# B&R Automation Studio project Kontrol (part 3)

#### Cyclic.st
```iecst
PROGRAM _CYCLIC

    IF NOT PgsTagValid(TagManager.ident) THEN
        RETURN;
    END_IF

	cm0985Meter();

    phaseFault(
        Enable  := TRUE,
        Ph1     := cm0985Meter.Ug1,
        Ph2     := cm0985Meter.Ug2,
        Ph3     := cm0985Meter.Ug3
    );

(*******************************************************
****************** Circuit Breaker  ********************
*******************************************************)
    avr.DigInputs.Online := CB52.st.closed;
    gov.DigInputs.Online := CB52.st.closed;

(******************************************************)
    //Reset
    IF A65.di.reset THEN
        //A65.di.reset        := FALSE;
        avr.DigInputs.Reset := TRUE;
		gov.DigInputs.Reset := TRUE;
		//Reset to Auto Mode
		//gov.DigInputs.Auto  := TRUE;
		//avr.DigInputs.Auto  := TRUE;
    END_IF;

    IF NOT A65.di.remote THEN
        //GOV
        gov.DigInputs.Start     := A65.di.gov_enable;
        gov.DigInputs.Stop      := NOT A65.di.gov_enable;
        gov.DigInputs.Unload    := A65.di.gov_unload;
		gov.DigInputs.RefUp		:= A65.di.gov_up;
		gov.DigInputs.RefDown	:= A65.di.gov_down;
        IF A65.di.gov_ctrl_pwr_enable THEN
            gov.CtrlOnline  := PGS_GOV_CA_PWR;
        ELSE
            gov.CtrlOnline  := PGS_GOV_CA_HZ_1;
        END_IF;

        //AVR
		A65.di.avr_unload		:= A65.di.gov_unload;
        avr.DigInputs.Start     := A65.di.avr_enable;
        avr.DigInputs.Stop      := NOT A65.di.avr_enable;
        avr.DigInputs.Unload    := A65.di.avr_unload;
		avr.DigInputs.RefUp		:= A65.di.avr_ref_up;
		avr.DigInputs.RefDown	:= A65.di.avr_ref_down;

        IF A65.di.avr_ctrl_qm_enable    THEN
            avr.CtrlOnline  := PGS_AVR_CA_QM;
        ELSIF  A65.di.avr_ctrl_pf_enable THEN
            avr.CtrlOnline  := PGS_AVR_CA_PF;
        ELSE
            avr.CtrlOnline  := PGS_AVR_CA_UM_1;
        END_IF;

    END_IF;

    (******************************************************)

	//TRIP
	IF A65.di.avr_trip THEN
        avr.DigInputs.Stop := TRUE;
    END_IF;
    IF A65.di.gov_trip THEN
        gov.DigInputs.Stop := TRUE;
    END_IF;

	//Meters

    //Icc ==> fix 4-20mA
    scale_if.x1 := 4.0;
    scale_if.x2 := 20.0;
    if_input	:= IfAvg * 16.0 / 32767.0 + 4.0;

    scale_if(
        x   := if_input,
        y1  := SysPar.Gen.IfMin,
        y2  := SysPar.Gen.IfMax
    );
	meter.In.If := scale_if.y;

	//Vcc ==> fix 4-20mA
    scale_uf.x1 := 4.0;
    scale_uf.x2 := 20.0;
	uf_input	:= UfAvg * 16.0 / 32767.0 + 4.0;
    scale_uf(
        x   := uf_input,
        y1  := SysPar.Gen.UfMin,
        y2  := SysPar.Gen.UfMax
    );
	meter.In.Uf := scale_uf.y;

	filter_uf( x := meter.In.Uf );
    //Ub
    IF cm0985Main.Enable3phase THEN
        meter.In.Ub := (cm0985Meter.Un12 + cm0985Meter.Un23 + cm0985Meter.Un31) / 3;
    ELSE
        meter.In.Ub := cm0985Meter.Un12;
    END_IF;
	//Um
	IF NOT phaseFault.Fault1 AND NOT phaseFault.Fault2 AND NOT phaseFault.Fault3 THEN
        meter.In.Um 	:=  cm0985Meter.Ug;
    ELSIF phaseFault.Fault1 AND NOT phaseFault.Fault2 AND NOT phaseFault.Fault3 THEN
        meter.In.Um 	:=  cm0985Meter.Ug23;
    ELSIF NOT phaseFault.Fault1 AND phaseFault.Fault2 AND NOT phaseFault.Fault3 THEN
        meter.In.Um 	:=  cm0985Meter.Ug31;
    ELSIF NOT phaseFault.Fault1 AND NOT phaseFault.Fault2 AND phaseFault.Fault3 THEN
        meter.In.Um 	:=  cm0985Meter.Ug12;
    ELSE
        meter.In.Um     :=  phaseFault.Phm * SQRT(3);
    END_IF

	meter.In.Im		:= cm0985Meter.Ig;
	IF meter.In.Um < 5 THEN
		meter.In.Fm		:= 0.0;
		meter.In.PF		:= 1.0;
	ELSE
		meter.In.Fm		:= cm0985Meter.Fg;
		meter.In.PF		:= cm0985Meter.PFg;
	END_IF;
	meter.In.Pm		:= cm0985Meter.Pg;
	meter.In.Qm		:= cm0985Meter.Qg;
	meter.In.Sm		:= cm0985Meter.Sg;

    rpm1(ppr := REAL_TO_INT(SysPar.Gen.PPR1));
    filter_rpm1.IN := rpm1.Output;
	filter_rpm1();

    rpm2(ppr := REAL_TO_INT(SysPar.Gen.PPR2));
    IF SysPar.Gen.PPR2 <> 0 THEN
		filter_rpm2.IN := rpm2.Output;
	ELSE
		filter_rpm2.IN := 0.0;
	END_IF;
    filter_rpm2();

	IF filter_rpm1.OUT > filter_rpm2.OUT THEN
	    meter.In.Rot := filter_rpm1.OUT;
    ELSE
	    meter.In.Rot := filter_rpm2.OUT;
    END_IF;

	IF SysPar.Gen.PPR2 <> 0 THEN
		A65.do.rpm_fault := ( ABS(filter_rpm1.OUT - filter_rpm2.OUT) / meter.Base.Rot ) > 0.05;
	ELSE
		A65.do.rpm_fault := FALSE;
	END_IF;
	meter       ();

	//Position
    //pos1 - ==> fix 4-20mA
	pos1_input	    := INT_TO_REAL(A65.ai.pos1) * 16.0 / 32767.0 + 4.0;
	filter_pos1(IN:=pos1_input);
    scale_pos1(
        x   := filter_pos1.OUT,
		x1  := SysPar.Gen.Pos1_0p,
        x2  := SysPar.Gen.Pos1_100p
    );
	pos1.PosIn	:= scale_pos1.y;

    pos2_input	    := INT_TO_REAL(A65.ai.pos2) * 16.0 / 32767.0 + 4.0;
    scale_pos2(
        x   := pos2_input,
		x1  := SysPar.Gen.Pos2_0p,
		x2  := SysPar.Gen.Pos2_100p
	);
	pos2.PosIn	:= scale_pos2.y;

    pos3_input	    := INT_TO_REAL(A65.ai.pos3) * 16.0 / 32767.0 + 4.0;
    scale_pos3(
        x   := pos3_input,
		x1  := SysPar.Gen.Pos3_0p,
		x2  := SysPar.Gen.Pos3_100p
	);
    pos3.PosIn := scale_pos3.y;

	//Syncronizer
    IF A65.di.remote THEN
        cm0985IO.do.SyncSlip    := SysUpdate.EnableSync;
        cm0985IO.do.SyncDeadBus := SysUpdate.EnableDeadBus AND NOT SysUpdate.EnableSync;
    ELSE
        cm0985IO.do.SyncSlip    := A65.di.sync_enable AND NOT CB52.st.closed;
        cm0985IO.do.SyncDeadBus := A65.di.dead_bus_enable AND NOT CB52.st.closed AND NOT A65.di.sync_enable;
    END_IF;
	A65.do.sync_enabled     := cm0985IO.do.SyncSlip OR cm0985IO.do.SyncDeadBus;
    IF cm0985IO.do.SyncSlip THEN
		IF cm0985Meter.dAngle > 15 AND cm0985Meter.dAngle < 345 THEN
			gov.SetPoints.fastSetHz := (cm0985Meter.Fs1 / meter.Base.Fm) * 1.001;
		ELSE
			gov.SetPoints.fastSetHz := cm0985Meter.Fs1 / meter.Base.Fm;
		END_IF;
		avr.SetPoints.fastSetUm := meter.Out.Ub;
	END_IF;

//=======================================================================
//=====	Para maior estabilidade do controle de potência	=================
//=======================================================================
	// Filtro da leitura da potência para estabilizar o sinal
	IF meter.Out.Pm <> 0 THEN
		filter_pwr(IN:=meter.Out.Pm);
	ELSE
		filter_pwr(IN:=0.0001);
	END_IF;
	// Verifica se a diferença em módulo da potência é menor que 1.5%
	IF  ABS(filter_pwr.OUT - gov.SetPoints.fastSetPwr) < gov.Parameter.CtrlAuto.CaPwr.Kdp
		// Verifica se a diferença em módulo do controle é menor que 2%
	AND ABS(1 - gov.SetPoints.fastSetHz) < 0.02	THEN
		// Se a deadband do PID for diferente, aplica deadband
		IF gov.Parameter.CtrlAuto.CaPwr.PID.db <> gov.Parameter.CtrlAuto.CaPwr.Kdp THEN
			gov.Parameter.CtrlAuto.CaPwr.PID.Update		:= TRUE;
			gov.Parameter.CtrlAuto.CaPwr.PIDHz.Update	:= TRUE;
		END_IF;
		gov.Parameter.CtrlAuto.CaPwr.PID.db		:= gov.Parameter.CtrlAuto.CaPwr.Kdp;
		gov.Parameter.CtrlAuto.CaPwr.PIDHz.db	:= gov.Parameter.CtrlAuto.CaPwr.Kdp;
	ELSE
		// Se a deadband do PID for diferente, desaplica deadband
		IF gov.Parameter.CtrlAuto.CaPwr.PID.db <> 0.00 THEN
			gov.Parameter.CtrlAuto.CaPwr.PID.Update	:= TRUE;
			gov.Parameter.CtrlAuto.CaPwr.PIDHz.Update	:= TRUE;
		END_IF;
		gov.Parameter.CtrlAuto.CaPwr.PID.db		:= 0.00;
		gov.Parameter.CtrlAuto.CaPwr.PIDHz.db	:= 0.00;
	END_IF;

	pwr_tp(IN:= CB52.st.closed, PT:=T#2s);
	IF pwr_tp.Q THEN
		gov.SetPoints.fastSetPwr := 0.1;
	END_IF;
	pwr_ton(IN:= CB52.st.closed AND NOT pwr_mem, PT:= T#5s);
	IF pwr_ton.Q THEN
		pwr_mem := TRUE;
		gov.SetPoints.SetPwr := gov.Parameter.CtrlAuto.CaPwr.Ref;
	END_IF;
	IF NOT CB52.st.closed THEN
		pwr_mem := FALSE;
	END_IF;
//=======================================================================
//=======================================================================

	//GOV
	gov     ();

	//POS1
    curve1	( In := gov.Out);
    pos1	( In := curve1.Out, Enable := (gov.DigOutputs.Status.Enable	AND NOT A65.di.gov_trip)
									OR  pos1.Mode > PGS_POS_MD_AUTO
									OR	A65.di.enable_pos1 );
    //Gov Out1
    IF A65.di.gov_trip THEN
		scale_gov_o1.x := (pos1.Parameter.HCC.dbHigh + pos1.Parameter.HCC.dbLow) / 2.0;
    ELSE
        scale_gov_o1.x := pos1.Out;
    END_IF;
	scale_gov_o1(
		x1 := 0.0,
		x2 := 1.0,
		y1 := 0,
		y2 := 32767.0);
    A65.ao.pos1 := REAL_TO_INT(scale_gov_o1.y);

    //POS2
    curve2	( In := gov.Out );
    pos2	( In := curve2.Out, Enable := (gov.DigOutputs.Status.Enable AND NOT A65.di.gov_trip)
									OR  pos2.Mode <> PGS_POS_MD_AUTO
									OR	A65.di.enable_pos2 );

    //Gov Out2
    IF A65.di.gov_trip THEN
		scale_gov_o2.x := (pos2.Parameter.HCC.dbHigh + pos2.Parameter.HCC.dbLow) / 2.0;
    ELSE
        scale_gov_o2.x := pos2.Out;
    END_IF;
	scale_gov_o2(
		x1 := 0.0,
		x2 := 1.0,
		y1 := 0,
		y2 := 32767.0);
    A65.ao.pos2 := REAL_TO_INT(scale_gov_o2.y);

    //POS3
    curve3	( In := gov.Out );
    pos3	( In := curve3.Out, Enable := (gov.DigOutputs.Status.Enable AND NOT A65.di.gov_trip)
									OR  pos3.Mode <> PGS_POS_MD_AUTO
									OR	A65.di.enable_pos3 );
    //Gov Out3
    IF A65.di.gov_trip THEN
		scale_gov_o3.x := (pos3.Parameter.HCC.dbHigh + pos3.Parameter.HCC.dbLow) / 2.0;
    ELSE
        scale_gov_o3.x := pos3.Out;
    END_IF;
	scale_gov_o3(
		x1 := 0.0,
		x2 := 1.0,
		y1 := 0,
		y2 := 32767.0);
    A65.ao.pos3 := REAL_TO_INT(scale_gov_o3.y);

    //Gov Pos feedback
    gov.PosIn   := pos1.PosOut;

    //Digital Outputs
    A65.do.gov_on               := gov.DigOutputs.Status.Enable;
    A65.do.rotation_zero        := meter.Out.Rot <= 0.01; //gov.DigOutputs.Status.Stopped;
    A65.do.rotation_nominal     := gov.DigOutputs.Status.RotationOk;
    A65.do.rotation_brake       := gov.DigOutputs.Status.RotationBrake;
    A65.do.gov_unload           := gov.DigOutputs.Status.Unloaded;
    A65.do.gov_over_rotation    := gov.DigOutputs.Trip.OverRotation;
    A65.do.power_zero           := meter.Out.Pm < gov.Parameter.CtrlAuto.CaPwr.RefOpen;

	//AVR
    avr			();
    //Avr Out1
	scale_avr_o1(
		x  := avr.Out,
		x1 := 0.0,
		x2 := 1.0,
		y1 := 0,
		y2 := 32767.0);
    A65.ao.pwr := REAL_TO_INT(scale_avr_o1.y);

    //Digital Outputs
    A65.do.avr_on               := avr.DigOutputs.Status.Enable;
    A65.do.field_flash_on	    := avr.DigOutputs.Status.FieldFlashOn;
	A65.do.voltage_nominal      := avr.DigOutputs.Status.VoltageOK;
    A65.do.avr_force_crowbar    := A65.di.avr_trip OR NOT avr.DigOutputs.Status.Enable;
    A65.do.avr_limiter_on       := avr.DigOutputs.Alarm.LimiterMin OR avr.DigOutputs.Alarm.LimiterMax;

//***************************************************
//****************** Hour Meter  ********************
//***************************************************
	hour_running	( enable := meter.Out.Rot > 0 ); // Maybe put frequency too?
	hour_online		( enable := gov.DigInputs.Online OR avr.DigInputs.Online );

//***************************************************
//**************** Energy Meter  ********************
//***************************************************
	energy_active	(
		enable	:= TRUE,
		power	:= meter.In.Pm
	);
	energy_reactive	(
		enable	:= TRUE,
		power	:= meter.In.Qm
	);

END_PROGRAM
```

- Cyclic.st.bak (not shown)

- Init.st.bak (not shown)

- Variables.var.bak (not shown)

### Share.var
```iecst
(*Inputs*)
VAR
	Protection : PgsProtType;
END_VAR
(*Parameters*)
VAR
	ProtPar : PgsProtParType;
END_VAR
(*Outputs*)
VAR
	ProtFlag : PgsProtFlagType;
	ExcTemp : REAL;
END_VAR
```

### Program Logical/Kontrol/Protection/Protection (IEC)

#### Variables.var
```iecst
(*Excitation*)
VAR
	ExcPhaseFault : PgsProtPhaseFault;
	timer_crowbar : TON;
	LExc_Crowbar : PgsProgLatch;
	LExc_OverTemp : PgsProgLatch;
END_VAR
(*Phase Sequence Elements*)
VAR
	V0 : PgsProtSeq0;
	V1 : PgsProtSeq1;
	V2 : PgsProtSeq2;
	I0 : PgsProtSeq0;
	I1 : PgsProtSeq1;
	I2 : PgsProtSeq2;
END_VAR
(*timers*)
VAR
	ton_ugseq : TON;
	ton_igseq : TON;
	ton_ubseq : TON;
END_VAR
(*Latchs*)
VAR
	L86E : PgsProgLatch;
	L86H : PgsProgLatch;
END_VAR
(*Protection 59*)
VAR
	L59A_L1 : PgsProgLatch;
	L59B_L1 : PgsProgLatch;
	L59C_L1 : PgsProgLatch;
	L59AB_L1 : PgsProgLatch;
	L59BC_L1 : PgsProgLatch;
	L59CA_L1 : PgsProgLatch;
	L59V1_L1 : PgsProgLatch;
	L59Q_L1 : PgsProgLatch;
	L59G_L1 : PgsProgLatch;
	L59A_L2 : PgsProgLatch;
	L59B_L2 : PgsProgLatch;
	L59C_L2 : PgsProgLatch;
	L59AB_L2 : PgsProgLatch;
	L59BC_L2 : PgsProgLatch;
	L59CA_L2 : PgsProgLatch;
	L59V1_L2 : PgsProgLatch;
	L59Q_L2 : PgsProgLatch;
	L59G_L2 : PgsProgLatch;
END_VAR
(*Protection 27*)
VAR
	L27A_L1 : PgsProgLatch;
	L27B_L1 : PgsProgLatch;
	L27C_L1 : PgsProgLatch;
	L27AB_L1 : PgsProgLatch;
	L27BC_L1 : PgsProgLatch;
	L27CA_L1 : PgsProgLatch;
	L27V1_L1 : PgsProgLatch;
	L27A_L2 : PgsProgLatch;
	L27B_L2 : PgsProgLatch;
	L27C_L2 : PgsProgLatch;
	L27AB_L2 : PgsProgLatch;
	L27BC_L2 : PgsProgLatch;
	L27CA_L2 : PgsProgLatch;
	L27V1_L2 : PgsProgLatch;
END_VAR
(*Protection 81*)
VAR
	L81O_L1 : PgsProgLatch;
	L81O_L2 : PgsProgLatch;
	L81U_L1 : PgsProgLatch;
	L81U_L2 : PgsProgLatch;
END_VAR
(*Protection 32*)
VAR
	L32OP_L1 : PgsProgLatch;
	L32UP_L1 : PgsProgLatch;
	L32OQ_L1 : PgsProgLatch;
	L32UQ_L1 : PgsProgLatch;
END_VAR
(*Protection 24*)
VAR
	L24_L1 : PgsProgLatch;
END_VAR
(*Protection 40*)
VAR
	L40_L1 : PgsProgLatch;
	L40_L2 : PgsProgLatch;
END_VAR
(*Protection 50*)
VAR
	L50PA_L1 : PgsProgLatch;
	L50PB_L1 : PgsProgLatch;
	L50PC_L1 : PgsProgLatch;
	L50Q_L1 : PgsProgLatch;
	L50G_L1 : PgsProgLatch;
	L50PA_L2 : PgsProgLatch;
	L50PB_L2 : PgsProgLatch;
	L50PC_L2 : PgsProgLatch;
	L50Q_L2 : PgsProgLatch;
	L50G_L2 : PgsProgLatch;
END_VAR
(*Protection 51*)
VAR
	L51VA_L1 : PgsProgLatch;
	L51VB_L1 : PgsProgLatch;
	L51VC_L1 : PgsProgLatch;
	L51PA_L1 : PgsProgLatch;
	L51PB_L1 : PgsProgLatch;
	L51PC_L1 : PgsProgLatch;
	L51Q_L1 : PgsProgLatch;
	L51G_L1 : PgsProgLatch;
END_VAR
(*Event*)
(*
VAR
	EvtGroup : PgsEvtGroup;
END_VAR
VAR RETAIN
	EvtMemory : ARRAY[0..1999] OF USINT;
END_VAR
*)
```

#### Cyclic.st
```iecst
PROGRAM _CYCLIC

    IF NOT PgsTagValid(TagManager.ident) THEN
        RETURN;
    END_IF
	Protection.di.reset := A65.di.reset;

	//Generator Phase Fault
    ProtFlag.GenPhAFault    := phaseFault.Fault1;
    ProtFlag.GenPhBFault    := phaseFault.Fault2;
    ProtFlag.GenPhCFault    := phaseFault.Fault3;

    //Phase Sequency Fault
	ton_ugseq(IN:=cm0985IO.di.UgPhSeqFault 	AND meter.Out.Um > 0.5, PT:=T#5s);
	ton_igseq(IN:=cm0985IO.di.IgPhSeqFault 	AND meter.Out.Im > 0.1, PT:=T#5s);
	ton_ubseq(IN:=cm0985IO.di.Us1PhSeqFault	AND meter.Out.Ub > 0.5, PT:=T#5s);
	ProtFlag.UgPhSeqFault		:= ton_ugseq.Q;
	ProtFlag.IgPhSeqFault		:= ton_igseq.Q;
	ProtFlag.Us1PhSeqFault		:= ton_ubseq.Q;

    //Power Excitation Phase Fault
    ExcPhaseFault(
        Enable  :=  meter.Out.Um > 0.5,
        Ph1     := cm0985Meter.Ub1,
        Ph2     := cm0985Meter.Ub2,
        Ph3     := cm0985Meter.Ub3
    );
    ProtFlag.ExcPhAFault    := ExcPhaseFault.Fault1;
    ProtFlag.ExcPhBFault    := ExcPhaseFault.Fault2;
    ProtFlag.ExcPhCFault    := ExcPhaseFault.Fault3;

	// Analog Temperature
    ExcTemp := INT_TO_REAL(Protection.ai.ExcTemp)/ 10.0;

    // Sensor Rotation Fault
    ProtFlag.RpmFault   := A65.do.rpm_fault;

	//Excitation
	timer_crowbar(IN:=avr.DigOutputs.Status.Enable AND NOT Protection.di.crowbar_ok, PT:=T#1s);
	LExc_Crowbar( Reset := Protection.di.reset, In := timer_crowbar.Q );
	ProtFlag.ExcCrowBar			:= LExc_Crowbar.Out;
	LExc_OverTemp( Reset := Protection.di.reset, In :=  NOT Protection.di.pwr_temp_ok OR ExcTemp	> 90.0 );
	ProtFlag.ExcOverTemp		:= LExc_OverTemp.Out;

	//Voltage Sequence Elements
	V0(
        PhaseA := cm0985Meter.Ug1, AngleA := cm0985Meter.Ug1Angle,
        PhaseB := cm0985Meter.Ug2, AngleB := cm0985Meter.Ug2Angle,
        PhaseC := cm0985Meter.Ug3, AngleC := cm0985Meter.Ug3Angle
    );
	V1(
        ClockWise := cm0985.ClockWise,
        PhaseA := cm0985Meter.Ug1, AngleA := cm0985Meter.Ug1Angle,
        PhaseB := cm0985Meter.Ug2, AngleB := cm0985Meter.Ug2Angle,
        PhaseC := cm0985Meter.Ug3, AngleC := cm0985Meter.Ug3Angle
    );
	V2(
        ClockWise := cm0985.ClockWise,
        PhaseA := cm0985Meter.Ug1, AngleA := cm0985Meter.Ug1Angle,
        PhaseB := cm0985Meter.Ug2, AngleB := cm0985Meter.Ug2Angle,
        PhaseC := cm0985Meter.Ug3, AngleC := cm0985Meter.Ug3Angle
    );
	//Current Sequence Elements
    I0(
        PhaseA := cm0985Meter.Ig1, AngleA := cm0985Meter.Ig1Angle,
        PhaseB := cm0985Meter.Ig2, AngleB := cm0985Meter.Ig2Angle,
        PhaseC := cm0985Meter.Ig3, AngleC := cm0985Meter.Ig3Angle
    );
	I1(
        ClockWise := cm0985.ClockWise,
        PhaseA := cm0985Meter.Ig1, AngleA := cm0985Meter.Ig1Angle,
        PhaseB := cm0985Meter.Ig2, AngleB := cm0985Meter.Ig2Angle,
        PhaseC := cm0985Meter.Ig3, AngleC := cm0985Meter.Ig3Angle
    );
	I2(
        ClockWise := cm0985.ClockWise,
        PhaseA := cm0985Meter.Ig1, AngleA := cm0985Meter.Ig1Angle,
        PhaseB := cm0985Meter.Ig2, AngleB := cm0985Meter.Ig2Angle,
        PhaseC := cm0985Meter.Ig3, AngleC := cm0985Meter.Ig3Angle
    );

	// Phase Overvoltage Level 1
	P59A_L1( Enable := P59A_L1.Parameter.Level <> 0.0, In := cm0985Meter.Ug1 );
	P59B_L1( Enable := P59B_L1.Parameter.Level <> 0.0, In := cm0985Meter.Ug2 );
	P59C_L1( Enable := P59C_L1.Parameter.Level <> 0.0, In := cm0985Meter.Ug3 );
	L59A_L1( Reset := Protection.di.reset, In := P59A_L1.O62T );
	L59B_L1( Reset := Protection.di.reset, In := P59B_L1.O62T );
	L59C_L1( Reset := Protection.di.reset, In := P59C_L1.O62T );
	// Phase Overvoltage Level 2
	P59A_L2( Enable := P59A_L2.Parameter.Level <> 0.0, In := cm0985Meter.Ug1 );
	P59B_L2( Enable := P59B_L2.Parameter.Level <> 0.0, In := cm0985Meter.Ug2 );
	P59C_L2( Enable := P59C_L2.Parameter.Level <> 0.0, In := cm0985Meter.Ug3 );
	L59A_L2( Reset := Protection.di.reset, In := P59A_L2.O62T );
	L59B_L2( Reset := Protection.di.reset, In := P59B_L2.O62T );
	L59C_L2( Reset := Protection.di.reset, In := P59C_L2.O62T );
	// Phase-Phase Overvoltage Level 1
	P59AB_L1( Enable := P59AB_L1.Parameter.Level <> 0.0, In := cm0985Meter.Ug12 );
	P59BC_L1( Enable := P59BC_L1.Parameter.Level <> 0.0, In := cm0985Meter.Ug23 );
	P59CA_L1( Enable := P59CA_L1.Parameter.Level <> 0.0, In := cm0985Meter.Ug31 );
	L59AB_L1( Reset := Protection.di.reset, In := P59AB_L1.O62T );
	L59BC_L1( Reset := Protection.di.reset, In := P59BC_L1.O62T );
	L59CA_L1( Reset := Protection.di.reset, In := P59CA_L1.O62T );
	// Phase-Phase Overvoltage Level 2
	P59AB_L2( Enable := P59AB_L2.Parameter.Level <> 0.0, In := cm0985Meter.Ug12 );
	P59BC_L2( Enable := P59BC_L2.Parameter.Level <> 0.0, In := cm0985Meter.Ug23 );
	P59CA_L2( Enable := P59CA_L2.Parameter.Level <> 0.0, In := cm0985Meter.Ug31 );
	L59AB_L2( Reset := Protection.di.reset, In := P59AB_L2.O62T );
	L59BC_L2( Reset := Protection.di.reset, In := P59BC_L2.O62T );
	L59CA_L2( Reset := Protection.di.reset, In := P59CA_L2.O62T );
	// Positive Sequence Overvoltage Level 1
	P59V1_L1( Enable := P59V1_L1.Parameter.Level <> 0.0, In := V1.Phase1 );
	L59V1_L1( Reset := Protection.di.reset, In := P59V1_L1.O62T );
	// Positive Sequence Overvoltage Level 2
	P59V1_L2( Enable := P59V1_L2.Parameter.Level <> 0.0, In := V1.Phase1 );
	L59V1_L2( Reset := Protection.di.reset, In := P59V1_L2.O62T );
	// Negative Sequence Overvoltage Level 1
	P59Q_L1( Enable := P59Q_L1.Parameter.Level <> 0.0, In := V2.Phase2 );
	L59Q_L1( Reset := Protection.di.reset, In := P59Q_L1.O62T );
	// Negative Sequence Overvoltage Level 2
	P59Q_L2( Enable := P59Q_L2.Parameter.Level <> 0.0, In := V2.Phase2 );
	L59Q_L2( Reset := Protection.di.reset, In := P59Q_L2.O62T );
	// Zero Sequence Overvoltage Level 1
	P59G_L1( Enable := P59G_L1.Parameter.Level <> 0.0, In := V0.Phase0 );
	L59G_L1( Reset := Protection.di.reset, In := P59G_L1.O62T );
	// Zero Sequence Overvoltage Level 2
	P59G_L2( Enable := P59G_L2.Parameter.Level <> 0.0, In := V0.Phase0 );
	L59G_L2( Reset := Protection.di.reset, In := P59G_L2.O62T );

	// Phase Undervoltage Level 1
	P27A_L1( Enable := P27A_L1.Parameter.Level <> 0.0 AND CB52.st.closed, In := cm0985Meter.Ug1 );
	P27B_L1( Enable := P27B_L1.Parameter.Level <> 0.0 AND CB52.st.closed, In := cm0985Meter.Ug2 );
	P27C_L1( Enable := P27C_L1.Parameter.Level <> 0.0 AND CB52.st.closed, In := cm0985Meter.Ug3 );
	L27A_L1( Reset := Protection.di.reset, In := P27A_L1.O62T );
	L27B_L1( Reset := Protection.di.reset, In := P27B_L1.O62T );
	L27C_L1( Reset := Protection.di.reset, In := P27C_L1.O62T );
	// Phase Undervoltage Level 2
	P27A_L2( Enable := P27A_L2.Parameter.Level <> 0.0 AND CB52.st.closed, In := cm0985Meter.Ug1 );
	P27B_L2( Enable := P27B_L2.Parameter.Level <> 0.0 AND CB52.st.closed, In := cm0985Meter.Ug2 );
	P27C_L2( Enable := P27C_L2.Parameter.Level <> 0.0 AND CB52.st.closed, In := cm0985Meter.Ug3 );
	L27A_L2( Reset := Protection.di.reset, In := P27A_L2.O62T );
	L27B_L2( Reset := Protection.di.reset, In := P27B_L2.O62T );
	L27C_L2( Reset := Protection.di.reset, In := P27C_L2.O62T );
	// Phase-Phase Undervoltage Level 1
	P27AB_L1( Enable := P27AB_L1.Parameter.Level <> 0.0 AND CB52.st.closed, In := cm0985Meter.Ug12 );
	P27BC_L1( Enable := P27BC_L1.Parameter.Level <> 0.0 AND CB52.st.closed, In := cm0985Meter.Ug23 );
	P27CA_L1( Enable := P27CA_L1.Parameter.Level <> 0.0 AND CB52.st.closed, In := cm0985Meter.Ug31 );
	L27AB_L1( Reset := Protection.di.reset, In := P27AB_L1.O62T );
	L27BC_L1( Reset := Protection.di.reset, In := P27BC_L1.O62T );
	L27CA_L1( Reset := Protection.di.reset, In := P27CA_L1.O62T );
	// Phase-Phase Undervoltage Level 2
	P27AB_L2( Enable := P27AB_L2.Parameter.Level <> 0.0 AND CB52.st.closed, In := cm0985Meter.Ug12 );
	P27BC_L2( Enable := P27BC_L2.Parameter.Level <> 0.0 AND CB52.st.closed, In := cm0985Meter.Ug23 );
	P27CA_L2( Enable := P27CA_L2.Parameter.Level <> 0.0 AND CB52.st.closed, In := cm0985Meter.Ug31 );
	L27AB_L2( Reset := Protection.di.reset, In := P27AB_L2.O62T );
	L27BC_L2( Reset := Protection.di.reset, In := P27BC_L2.O62T );
	L27CA_L2( Reset := Protection.di.reset, In := P27CA_L2.O62T );
	// Positive Sequence Undervoltage Level 1
	P27V1_L1( Enable := P27V1_L1.Parameter.Level <> 0.0 AND CB52.st.closed, In := V1.Phase1 );
	L27V1_L1( Reset := Protection.di.reset, In := P27V1_L1.O62T );
	// Positive Sequence Undervoltage Level 2
	P27V1_L2( Enable := P27V1_L2.Parameter.Level <> 0.0 AND CB52.st.closed, In := V1.Phase1 );
	L27V1_L2( Reset := Protection.di.reset, In := P27V1_L2.O62T );

	// Overfrequency Level 1
	P81O_L1( Enable := P81O_L1.Parameter.Level <> 0.0 AND CB52.st.closed, In := meter.In.Fm );
	L81O_L1( Reset := Protection.di.reset, In := P81O_L1.O62T );
	// Overfrequency Level 2
	P81O_L2( Enable := P81O_L2.Parameter.Level <> 0.0 AND CB52.st.closed, In := meter.In.Fm );
	L81O_L2( Reset := Protection.di.reset, In := P81O_L2.O62T );

	// Underfrequency Level 1
	P81U_L1( Enable := P81U_L1.Parameter.Level <> 0.0 AND CB52.st.closed, In := meter.In.Fm );
	L81U_L1( Reset := Protection.di.reset, In := P81U_L1.O62T );
	// Underfrequency Level 2
	P81U_L2( Enable := P81U_L2.Parameter.Level <> 0.0 AND CB52.st.closed, In := meter.In.Fm );
	L81U_L2( Reset := Protection.di.reset, In := P81U_L2.O62T );

	// Over Active Power Level 1
	P32OP_L1( Enable := P32OP_L1.Parameter.Level <> 0.0, In := meter.Out.Pm );
	L32OP_L1( Reset := Protection.di.reset, In := P32OP_L1.O62T );
	// Under Active Power Level 1
	P32UP_L1( Enable := P32UP_L1.Parameter.Level <> 0.0, In := meter.Out.Pm );
	L32UP_L1( Reset := Protection.di.reset, In := P32UP_L1.O62T );

	// Over Reactive Power Level 1
	P32OQ_L1( Enable := P32OQ_L1.Parameter.Level <> 0.0, In := meter.Out.Qm );
	L32OQ_L1( Reset := Protection.di.reset, In := P32OQ_L1.O62T );
	// Under Reactive Power Level 1
	P32UQ_L1( Enable := P32UQ_L1.Parameter.Level <> 0.0, In := meter.Out.Qm );
	L32UQ_L1( Reset := Protection.di.reset, In := P32UQ_L1.O62T );

	// Phase Instantaneous Overcurrent Level 1
	P50PA_L1( Enable := P50PA_L1.Parameter.Level <> 0.0, In := cm0985Meter.Ig1 );
	P50PB_L1( Enable := P50PB_L1.Parameter.Level <> 0.0, In := cm0985Meter.Ig2 );
	P50PC_L1( Enable := P50PC_L1.Parameter.Level <> 0.0, In := cm0985Meter.Ig3 );
	L50PA_L1( Reset := Protection.di.reset, In := P50PA_L1.O62T );
	L50PB_L1( Reset := Protection.di.reset, In := P50PB_L1.O62T );
	L50PC_L1( Reset := Protection.di.reset, In := P50PC_L1.O62T );
	// Negative Sequence Instantaneous Overcurrent Level 1
	P50Q_L1 ( Enable := P50Q_L1.Parameter.Level <> 0.0, In := I2.Phase2 );
	L50Q_L1( Reset := Protection.di.reset, In := P50Q_L1.O62T );
	// Residual Instantaneous Overcurrent Level 1
	P50G_L1 ( Enable := P50G_L1.Parameter.Level <> 0.0, In := I0.Phase0 );
	L50G_L1( Reset := Protection.di.reset, In := P50G_L1.O62T );
	// Phase Instantaneous Overcurrent Level 2
	P50PA_L2( Enable := P50PA_L2.Parameter.Level <> 0.0, In := cm0985Meter.Ig1 );
	P50PB_L2( Enable := P50PB_L2.Parameter.Level <> 0.0, In := cm0985Meter.Ig2 );
	P50PC_L2( Enable := P50PC_L2.Parameter.Level <> 0.0, In := cm0985Meter.Ig3 );
	L50PA_L2( Reset := Protection.di.reset, In := P50PA_L2.O62T );
	L50PB_L2( Reset := Protection.di.reset, In := P50PB_L2.O62T );
	L50PC_L2( Reset := Protection.di.reset, In := P50PC_L2.O62T );
	// Negative Sequence Instantaneous Overcurrent Level 2
	P50Q_L2 ( Enable := P50Q_L2.Parameter.Level <> 0.0, In := I2.Phase2 );
	L50Q_L2( Reset := Protection.di.reset, In := P50Q_L2.O62T );
	// Residual Instantaneous Overcurrent Level 2
	P50G_L2 ( Enable := P50G_L2.Parameter.Level <> 0.0, In := I0.Phase0 );
	L50G_L2( Reset := Protection.di.reset, In := P50G_L2.O62T );

	// Voltage Restraint Time Overcurrent - 51V
	P51VA_L1( Enable := TRUE, I := cm0985Meter.Ig1, V := cm0985Meter.Ug1 );
	P51VB_L1( Enable := TRUE, I := cm0985Meter.Ig2, V := cm0985Meter.Ug2 );
	P51VC_L1( Enable := TRUE, I := cm0985Meter.Ig3, V := cm0985Meter.Ug3 );
	L51VA_L1( Reset := Protection.di.reset, In := P51VA_L1.O51VT );
	L51VB_L1( Reset := Protection.di.reset, In := P51VB_L1.O51VT );
	L51VC_L1( Reset := Protection.di.reset, In := P51VC_L1.O51VT );
	// Phase Time Overcurrent - 51P
	P51PA_L1( Enable := TRUE, I := cm0985Meter.Ig1 );
	P51PB_L1( Enable := TRUE, I := cm0985Meter.Ig2 );
	P51PC_L1( Enable := TRUE, I := cm0985Meter.Ig3 );
	L51PA_L1( Reset := Protection.di.reset, In := P51PA_L1.O51VT );
	L51PB_L1( Reset := Protection.di.reset, In := P51PB_L1.O51VT );
	L51PC_L1( Reset := Protection.di.reset, In := P51PC_L1.O51VT );
	// Negative Sequence Time Overcurrent - 51Q
	P51Q_L1( Enable := TRUE, I := I2.Phase2 );
	L51Q_L1( Reset := Protection.di.reset, In := P51Q_L1.O51VT );
	// Residual Time Overcurrent - 51Q
	P51G_L1( Enable := TRUE, I := I0.Phase0 );
	L51G_L1( Reset := Protection.di.reset, In := P51G_L1.O51VT );

	// V/Hz Element - 24
	P24_L1( Enable := P24_L1.Parameter.VHZ <> 0.0, V := meter.In.Um, Hz:= meter.In.Fm );
    L24_L1( Reset := Protection.di.reset, In := P24_L1.O24T );

   	IF I1.Phase1 > 0.0 THEN
		// Loss of Field Level 1 - 40
		P40_L1( Enable := P40_L1.Parameter.diameter <> 0.0, Zmodule := V1.Phase1/I1.Phase1, Zangle := V1.Angle1 - I1.Angle1 );
		// Loss of Field Level 2 - 40
		P40_L2( Enable := P40_L2.Parameter.diameter <> 0.0, Zmodule := V1.Phase1/I1.Phase1, Zangle := V1.Angle1 - I1.Angle1 );
	ELSE
		P40_L1( Enable := FALSE );
		P40_L2( Enable := FALSE );
	END_IF;
	L40_L1( Reset := Protection.di.reset, In := P40_L1.O40ZT );
	L40_L2( Reset := Protection.di.reset, In := P40_L2.O40ZT );

    //86H
	L86H(
		Reset	:= Protection.di.reset,
		In		:=
			ProtFlag.WatchDog					OR
			gov.DigOutputs.Trip.Trip			OR
			pos1.Trip							OR
			pos2.Trip							OR
			pos3.Trip
	);

	//86E
	L86E(
		Reset	:= Protection.di.reset,
		In		:=
			//59P
			P59A_L1.O62T OR P59B_L1.O62T OR P59C_L1.O62T OR
			P59A_L2.O62T OR P59B_L2.O62T OR P59C_L2.O62T OR
			//59PP
			P59AB_L1.O62T OR P59BC_L1.O62T OR P59CA_L1.O62T OR
			P59AB_L2.O62T OR P59BC_L2.O62T OR P59CA_L2.O62T OR
			//59Q
			P59Q_L1.O62T OR P59Q_L2.O62T OR
			//59G
			P59G_L1.O62T OR P59G_L2.O62T OR
			//59V1
			P59V1_L1.O62T OR P59V1_L2.O62T OR
			//27P
			P27A_L1.O62T OR P27B_L1.O62T OR P27C_L1.O62T OR
			P27A_L2.O62T OR P27B_L2.O62T OR P27C_L2.O62T OR
			//27PP
			P27AB_L1.O62T OR P27BC_L1.O62T OR P27CA_L1.O62T OR
			P27AB_L2.O62T OR P27BC_L2.O62T OR P27CA_L2.O62T OR
			//27V1
			P27V1_L1.O62T OR P27V1_L2.O62T OR
			//81O
			P81O_L1.O62T OR P81O_L2.O62T OR
			//81U
			P81U_L1.O62T OR P81U_L2.O62T OR
			//32
			P32OP_L1.O62T OR P32UP_L1.O62T OR P32OQ_L1.O62T OR P32UQ_L1.O62T OR
			//50P
			P50PA_L1.O62T OR P50PB_L1.O62T OR P50PC_L1.O62T OR
			P50PA_L2.O62T OR P50PB_L2.O62T OR P50PC_L2.O62T OR
			//50Q
			P50Q_L1.O62T OR P50Q_L2.O62T OR
			//50G
			P50G_L1.O62T OR P50G_L2.O62T OR
			//51V
			P51VA_L1.O51VT OR P51VB_L1.O51VT OR P51VC_L1.O51VT OR
			//51P
			P51PA_L1.O51VT OR P51PB_L1.O51VT OR P51PC_L1.O51VT OR
			//51Q
			P51Q_L1.O51VT OR
			//51G
			P51G_L1.O51VT OR
			//24
			P24_L1.O24T OR
			//40
			P40_L1.O40ZT OR P40_L2.O40ZT OR
			//External Inputs
			ProtFlag.WatchDog					OR
			ProtFlag.ExcCrowBar					OR
			ProtFlag.ExcOverTemp				OR
			//AVR
			avr.DigOutputs.Trip.Trip			OR
			//GOV
			gov.DigOutputs.Trip.Trip			OR
			//86H
			L86H.Out
	);

	ProtFlag.T86H	:= L86H.Out;
	ProtFlag.T86E	:= L86E.Out;

    //TRIP
    Protection.do.trip_86e  := NOT L86E.Out;
	Protection.do.trip_86h  := NOT L86H.Out;

	P50BF.Parameter.Inom	:= meter.Base.Im;
	P50BF.Parameter.Time	:= ProtPar.T50BF;
	P50BF.I1				:= I1.Phase1;
	P50BF.I2				:= I2.Phase2;
    P50BF.Closed			:= CB52.st.closed;
    P50BF( Enable := TRUE, Trip := ProtFlag.T86E OR ProtFlag.T86H );

	Protection.do.trip_50bf := P50BF.O50BFT;

	/////////////
	/// FLAGS ///
	/////////////
	//59P
	ProtFlag.P59A_L1	:= P59A_L1.O62;
	ProtFlag.T59A_L1	:= P59A_L1.O62T;
	ProtFlag.L59A_L1	:= L59A_L1.Out;
	ProtFlag.P59B_L1	:= P59B_L1.O62;
	ProtFlag.T59B_L1	:= P59B_L1.O62T;
	ProtFlag.L59B_L1	:= L59B_L1.Out;
	ProtFlag.P59C_L1	:= P59C_L1.O62;
	ProtFlag.T59C_L1	:= P59C_L1.O62T;
	ProtFlag.L59C_L1	:= L59C_L1.Out;
	ProtFlag.P59A_L2	:= P59A_L2.O62;
	ProtFlag.T59A_L2	:= P59A_L2.O62T;
	ProtFlag.L59A_L2	:= L59A_L2.Out;
	ProtFlag.P59B_L2	:= P59B_L2.O62;
	ProtFlag.T59B_L2	:= P59B_L2.O62T;
	ProtFlag.L59B_L2	:= L59B_L2.Out;
	ProtFlag.P59C_L2	:= P59C_L2.O62;
	ProtFlag.T59C_L2	:= P59C_L2.O62T;
	ProtFlag.L59C_L2	:= L59C_L2.Out;
	//59PP
	ProtFlag.P59AB_L1	:= P59AB_L1.O62;
	ProtFlag.T59AB_L1	:= P59AB_L1.O62T;
	ProtFlag.L59AB_L1	:= L59AB_L1.Out;
	ProtFlag.P59BC_L1	:= P59BC_L1.O62;
	ProtFlag.T59BC_L1	:= P59BC_L1.O62T;
	ProtFlag.L59BC_L1	:= L59BC_L1.Out;
	ProtFlag.P59CA_L1	:= P59CA_L1.O62;
	ProtFlag.T59CA_L1	:= P59CA_L1.O62T;
	ProtFlag.L59CA_L1	:= L59CA_L1.Out;
	ProtFlag.P59AB_L2	:= P59AB_L2.O62;
	ProtFlag.T59AB_L2	:= P59AB_L2.O62T;
	ProtFlag.L59AB_L2	:= L59AB_L2.Out;
	ProtFlag.P59BC_L2	:= P59BC_L2.O62;
	ProtFlag.T59BC_L2	:= P59BC_L2.O62T;
	ProtFlag.L59BC_L2	:= L59BC_L2.Out;
	ProtFlag.P59CA_L2	:= P59CA_L2.O62;
	ProtFlag.T59CA_L2	:= P59CA_L2.O62T;
	ProtFlag.L59CA_L2	:= L59CA_L2.Out;
	//59Q
	ProtFlag.P59Q_L1	:= P59Q_L1.O62;
	ProtFlag.T59Q_L1	:= P59Q_L1.O62T;
	ProtFlag.L59Q_L1	:= L59Q_L1.Out;
	ProtFlag.P59Q_L2	:= P59Q_L2.O62;
	ProtFlag.T59Q_L2	:= P59Q_L2.O62T;
	ProtFlag.L59Q_L2	:= L59Q_L2.Out;
	//59G
	ProtFlag.P59G_L1	:= P59G_L1.O62;
	ProtFlag.T59G_L1	:= P59G_L1.O62T;
	ProtFlag.L59G_L1	:= L59G_L1.Out;
	ProtFlag.P59G_L2	:= P59G_L2.O62;
	ProtFlag.T59G_L2	:= P59G_L2.O62T;
	ProtFlag.L59G_L2	:= L59G_L2.Out;
	//59V1
	ProtFlag.P59V1_L1	:= P59V1_L1.O62;
	ProtFlag.T59V1_L1	:= P59V1_L1.O62T;
	ProtFlag.L59V1_L1	:= L59V1_L1.Out;
	ProtFlag.P59V1_L2	:= P59V1_L2.O62;
	ProtFlag.T59V1_L2	:= P59V1_L2.O62T;
	ProtFlag.L59V1_L2	:= L59V1_L2.Out;
	//27P
	ProtFlag.P27A_L1	:= P27A_L1.O62;
	ProtFlag.T27A_L1	:= P27A_L1.O62T;
	ProtFlag.L27A_L1	:= L27A_L1.Out;
	ProtFlag.P27B_L1	:= P27B_L1.O62;
	ProtFlag.T27B_L1	:= P27B_L1.O62T;
	ProtFlag.L27B_L1	:= L27B_L1.Out;
	ProtFlag.P27C_L1	:= P27C_L1.O62;
	ProtFlag.T27C_L1	:= P27C_L1.O62T;
	ProtFlag.L27C_L1	:= L27C_L1.Out;
	ProtFlag.P27A_L2	:= P27A_L2.O62;
	ProtFlag.T27A_L2	:= P27A_L2.O62T;
	ProtFlag.L27A_L2	:= L27A_L2.Out;
	ProtFlag.P27B_L2	:= P27B_L2.O62;
	ProtFlag.T27B_L2	:= P27B_L2.O62T;
	ProtFlag.L27B_L2	:= L27B_L2.Out;
	ProtFlag.P27C_L2	:= P27C_L2.O62;
	ProtFlag.T27C_L2	:= P27C_L2.O62T;
	ProtFlag.L27C_L2	:= L27C_L2.Out;
	//27PP
	ProtFlag.P27AB_L1	:= P27AB_L1.O62;
	ProtFlag.T27AB_L1	:= P27AB_L1.O62T;
	ProtFlag.L27AB_L1	:= L27AB_L1.Out;
	ProtFlag.P27BC_L1	:= P27BC_L1.O62;
	ProtFlag.T27BC_L1	:= P27BC_L1.O62T;
	ProtFlag.L27BC_L1	:= L27BC_L1.Out;
	ProtFlag.P27CA_L1	:= P27CA_L1.O62;
	ProtFlag.T27CA_L1	:= P27CA_L1.O62T;
	ProtFlag.L27CA_L1	:= L27CA_L1.Out;
	ProtFlag.P27AB_L2	:= P27AB_L2.O62;
	ProtFlag.T27AB_L2	:= P27AB_L2.O62T;
	ProtFlag.L27AB_L2	:= L27AB_L2.Out;
	ProtFlag.P27BC_L2	:= P27BC_L2.O62;
	ProtFlag.T27BC_L2	:= P27BC_L2.O62T;
	ProtFlag.L27BC_L2	:= L27BC_L2.Out;
	ProtFlag.P27CA_L2	:= P27CA_L2.O62;
	ProtFlag.T27CA_L2	:= P27CA_L2.O62T;
	ProtFlag.L27CA_L2	:= L27CA_L2.Out;
	//27V1
	ProtFlag.P27V1_L1	:= P27V1_L1.O62;
	ProtFlag.T27V1_L1	:= P27V1_L1.O62T;
	ProtFlag.L27V1_L1	:= L27V1_L1.Out;
	ProtFlag.P27V1_L2	:= P27V1_L2.O62;
	ProtFlag.T27V1_L2	:= P27V1_L2.O62T;
	ProtFlag.L27V1_L2	:= L27V1_L2.Out;
	//81O
	ProtFlag.P81O_L1	:= P81O_L1.O62;
	ProtFlag.T81O_L1	:= P81O_L1.O62T;
	ProtFlag.L81O_L1	:= L81O_L1.Out;
	ProtFlag.P81O_L2	:= P81O_L2.O62;
	ProtFlag.T81O_L2	:= P81O_L2.O62T;
	ProtFlag.L81O_L2	:= L81O_L2.Out;
	//81U
	ProtFlag.P81U_L1	:= P81U_L1.O62;
	ProtFlag.T81U_L1	:= P81U_L1.O62T;
	ProtFlag.L81U_L1	:= L81U_L1.Out;
	ProtFlag.P81U_L2	:= P81U_L2.O62;
	ProtFlag.T81U_L2	:= P81U_L2.O62T;
	ProtFlag.L81U_L2	:= L81U_L2.Out;
	//32OP
	ProtFlag.P32OP_L1	:= P32OP_L1.O62;
	ProtFlag.T32OP_L1	:= P32OP_L1.O62T;
	ProtFlag.L32OP_L1	:= L32OP_L1.Out;
	//32UP
	ProtFlag.P32UP_L1	:= P32UP_L1.O62;
	ProtFlag.T32UP_L1	:= P32UP_L1.O62T;
	ProtFlag.L32UP_L1	:= L32UP_L1.Out;
	//32OQ
	ProtFlag.P32OQ_L1	:= P32OQ_L1.O62;
	ProtFlag.T32OQ_L1	:= P32OQ_L1.O62T;
	ProtFlag.L32OQ_L1	:= L32OQ_L1.Out;
	//32UQ
	ProtFlag.P32UQ_L1	:= P32UQ_L1.O62;
	ProtFlag.T32UQ_L1	:= P32UQ_L1.O62T;
	ProtFlag.L32UQ_L1	:= L32UQ_L1.Out;
	//24
	ProtFlag.P24_L1	:= P24_L1.O24;
	ProtFlag.T24_L1	:= P24_L1.O24T;
	ProtFlag.L24_L1	:= L24_L1.Out;
	//40
	ProtFlag.P40_L1	:= P40_L1.O40Z;
	ProtFlag.T40_L1	:= P40_L1.O40ZT;
	ProtFlag.L40_L1	:= L40_L1.Out;
	ProtFlag.P40_L2	:= P40_L2.O40Z;
	ProtFlag.T40_L2	:= P40_L2.O40ZT;
	ProtFlag.L40_L2	:= L40_L2.Out;
	//50P
	ProtFlag.P50PA_L1	:= P50PA_L1.O62;
	ProtFlag.T50PA_L1	:= P50PA_L1.O62T;
	ProtFlag.L50PA_L1	:= L50PA_L1.Out;
	ProtFlag.P50PB_L1	:= P50PB_L1.O62;
	ProtFlag.T50PB_L1	:= P50PB_L1.O62T;
	ProtFlag.L50PB_L1	:= L50PB_L1.Out;
	ProtFlag.P50PC_L1	:= P50PC_L1.O62;
	ProtFlag.T50PC_L1	:= P50PC_L1.O62T;
	ProtFlag.L50PC_L1	:= L50PC_L1.Out;
	ProtFlag.P50PA_L2	:= P50PA_L2.O62;
	ProtFlag.T50PA_L2	:= P50PA_L2.O62T;
	ProtFlag.L50PA_L2	:= L50PA_L2.Out;
	ProtFlag.P50PB_L2	:= P50PB_L2.O62;
	ProtFlag.T50PB_L2	:= P50PB_L2.O62T;
	ProtFlag.L50PB_L2	:= L50PB_L2.Out;
	ProtFlag.P50PC_L2	:= P50PC_L2.O62;
	ProtFlag.T50PC_L2	:= P50PC_L2.O62T;
	ProtFlag.L50PC_L2	:= L50PC_L2.Out;
	//50Q
	ProtFlag.P50Q_L1	:= P50Q_L1.O62;
	ProtFlag.T50Q_L1	:= P50Q_L1.O62T;
	ProtFlag.L50Q_L1	:= L50Q_L1.Out;
	ProtFlag.P50Q_L2	:= P50Q_L2.O62;
	ProtFlag.T50Q_L2	:= P50Q_L2.O62T;
	ProtFlag.L50Q_L2	:= L50Q_L2.Out;
	//50G
	ProtFlag.P50G_L1	:= P50G_L1.O62;
	ProtFlag.T50G_L1	:= P50G_L1.O62T;
	ProtFlag.L50G_L1	:= L50G_L1.Out;
	ProtFlag.P50G_L2	:= P50G_L2.O62;
	ProtFlag.T50G_L2	:= P50G_L2.O62T;
	ProtFlag.L50G_L2	:= L50G_L2.Out;
	//51V
	ProtFlag.P51VA_L1	:= P51VA_L1.O51V;
	ProtFlag.T51VA_L1	:= P51VA_L1.O51VT;
	ProtFlag.R51VA_L1	:= P51VA_L1.O51VR;
	ProtFlag.L51VA_L1	:= L51VA_L1.Out;
	ProtFlag.P51VB_L1	:= P51VB_L1.O51V;
	ProtFlag.T51VB_L1	:= P51VB_L1.O51VT;
	ProtFlag.R51VB_L1	:= P51VB_L1.O51VR;
	ProtFlag.L51VB_L1	:= L51VB_L1.Out;
	ProtFlag.P51VC_L1	:= P51VC_L1.O51V;
	ProtFlag.T51VC_L1	:= P51VC_L1.O51VT;
	ProtFlag.R51VC_L1	:= P51VC_L1.O51VR;
	ProtFlag.L51VC_L1	:= L51VC_L1.Out;
	//51P
	ProtFlag.P51PA_L1	:= P51PA_L1.O51V;
	ProtFlag.T51PA_L1	:= P51PA_L1.O51VT;
	ProtFlag.R51PA_L1	:= P51PA_L1.O51VR;
	ProtFlag.L51PA_L1	:= L51PA_L1.Out;
	ProtFlag.P51PB_L1	:= P51PB_L1.O51V;
	ProtFlag.T51PB_L1	:= P51PB_L1.O51VT;
	ProtFlag.R51PB_L1	:= P51PB_L1.O51VR;
	ProtFlag.L51PB_L1	:= L51PB_L1.Out;
	ProtFlag.P51PC_L1	:= P51PC_L1.O51V;
	ProtFlag.T51PC_L1	:= P51PC_L1.O51VT;
	ProtFlag.R51PC_L1	:= P51PC_L1.O51VR;
	ProtFlag.L51PC_L1	:= L51PC_L1.Out;
	//51Q
	ProtFlag.P51Q_L1	:= P51Q_L1.O51V;
	ProtFlag.T51Q_L1	:= P51Q_L1.O51VT;
	ProtFlag.R51Q_L1	:= P51Q_L1.O51VR;
	ProtFlag.L51Q_L1	:= L51Q_L1.Out;
	//51G
	ProtFlag.P51G_L1	:= P51G_L1.O51V;
	ProtFlag.T51G_L1	:= P51G_L1.O51VT;
	ProtFlag.R51G_L1	:= P51G_L1.O51VR;
	ProtFlag.L51G_L1	:= L51G_L1.Out;

	/////////////
	/// RESET ///
	/////////////
	IF Protection.di.reset THEN
		Protection.di.reset	:= FALSE;
	END_IF;

//    EvtGroup( ident := Event );

END_PROGRAM
```

- Cyclic.st.bak (not shown)

- Init.st.bak (not shown)

### Program Logical/Kontrol/Protection/ProtUpdate (IEC)

#### Cyclic.st
```iecst
PROGRAM _CYCLIC
	IF SysUpdate.UpdateProt THEN
		SysUpdate.UpdateProt		:= FALSE;

		//59P
		P59A_L1.Parameter.Under		:= FALSE;
		P59A_L1.Parameter.Level		:= ProtPar.P59P_L1 * meter.Base.Um / SQRT(3.0);
		P59A_L1.Parameter.Time		:= ProtPar.T59P_L1;

		P59B_L1.Parameter := P59C_L1.Parameter := P59A_L1.Parameter;

		P59A_L2.Parameter.Under		:= FALSE;
		P59A_L2.Parameter.Level		:= ProtPar.P59P_L2 * meter.Base.Um / SQRT(3.0);
		P59A_L2.Parameter.Time		:= ProtPar.T59P_L2;

		P59B_L2.Parameter := P59C_L2.Parameter := P59A_L2.Parameter;

		//59PP
		P59AB_L1.Parameter.Under	:= FALSE;
		P59AB_L1.Parameter.Level	:= ProtPar.P59PP_L1 * meter.Base.Um;
		P59AB_L1.Parameter.Time		:= ProtPar.T59PP_L1;

		P59BC_L1.Parameter := P59CA_L1.Parameter := P59AB_L1.Parameter;

		P59AB_L2.Parameter.Under	:= FALSE;
		P59AB_L2.Parameter.Level	:= ProtPar.P59PP_L2 * meter.Base.Um;
		P59AB_L2.Parameter.Time		:= ProtPar.T59PP_L2;

		P59BC_L2.Parameter := P59CA_L2.Parameter := P59AB_L2.Parameter;

		//59Q
		P59Q_L1.Parameter.Under		:= FALSE;
		P59Q_L1.Parameter.Level		:= ProtPar.P59Q_L1 * meter.Base.Um / SQRT(3.0);
		P59Q_L1.Parameter.Time		:= ProtPar.T59Q_L1;

		P59Q_L2.Parameter.Under		:= FALSE;
		P59Q_L2.Parameter.Level		:= ProtPar.P59Q_L2 * meter.Base.Um / SQRT(3.0);
		P59Q_L2.Parameter.Time		:= ProtPar.T59Q_L2;

		//59G
		P59G_L1.Parameter.Under		:= FALSE;
		P59G_L1.Parameter.Level		:= ProtPar.P59G_L1 * meter.Base.Um / SQRT(3.0);
		P59G_L1.Parameter.Time		:= ProtPar.T59G_L1;

		P59G_L2.Parameter.Under		:= FALSE;
		P59G_L2.Parameter.Level		:= ProtPar.P59G_L2 * meter.Base.Um / SQRT(3.0);
		P59G_L2.Parameter.Time		:= ProtPar.T59G_L2;

		//59V1
		P59V1_L1.Parameter.Under	:= FALSE;
		P59V1_L1.Parameter.Level	:= ProtPar.P59V1_L1 * meter.Base.Um / SQRT(3.0);
		P59V1_L1.Parameter.Time		:= ProtPar.T59V1_L1;

		P59V1_L2.Parameter.Under	:= FALSE;
		P59V1_L2.Parameter.Level	:= ProtPar.P59V1_L2 * meter.Base.Um / SQRT(3.0);
		P59V1_L2.Parameter.Time		:= ProtPar.T59V1_L2;

		//27P
		P27A_L1.Parameter.Under		:= TRUE;
		P27A_L1.Parameter.Level		:= ProtPar.P27P_L1 * meter.Base.Um / SQRT(3.0);
		P27A_L1.Parameter.Time		:= ProtPar.T27P_L1;

		P27B_L1.Parameter := P27C_L1.Parameter := P27A_L1.Parameter;

		P27A_L2.Parameter.Under		:= TRUE;
		P27A_L2.Parameter.Level		:= ProtPar.P27P_L2 * meter.Base.Um / SQRT(3.0);
		P27A_L2.Parameter.Time		:= ProtPar.T27P_L2;

		P27B_L2.Parameter := P27C_L2.Parameter := P27A_L2.Parameter;

		//27PP
		P27AB_L1.Parameter.Under	:= TRUE;
		P27AB_L1.Parameter.Level	:= ProtPar.P27PP_L1 * meter.Base.Um;
		P27AB_L1.Parameter.Time		:= ProtPar.T27PP_L1;

		P27BC_L1.Parameter := P27CA_L1.Parameter := P27AB_L1.Parameter;

		P27AB_L2.Parameter.Under	:= TRUE;
		P27AB_L2.Parameter.Level	:= ProtPar.P27PP_L2 * meter.Base.Um;
		P27AB_L2.Parameter.Time		:= ProtPar.T27PP_L2;

		P27BC_L2.Parameter := P27CA_L2.Parameter := P27AB_L2.Parameter;

		//27V1
		P27V1_L1.Parameter.Under	:= TRUE;
		P27V1_L1.Parameter.Level	:= ProtPar.P27V1_L1 * meter.Base.Um / SQRT(3.0);
		P27V1_L1.Parameter.Time		:= ProtPar.T27V1_L1;

		P27V1_L2.Parameter.Under	:= TRUE;
		P27V1_L2.Parameter.Level	:= ProtPar.P27V1_L2 * meter.Base.Um / SQRT(3.0);
		P27V1_L2.Parameter.Time		:= ProtPar.T27V1_L2;

		//81O
		P81O_L1.Parameter.Under		:= FALSE;
		P81O_L1.Parameter.Level		:= ProtPar.P81O_L1 * meter.Base.Fm;
		P81O_L1.Parameter.Time		:= ProtPar.T81O_L1;

		P81O_L2.Parameter.Under		:= FALSE;
		P81O_L2.Parameter.Level		:= ProtPar.P81O_L2 * meter.Base.Fm;
		P81O_L2.Parameter.Time		:= ProtPar.T81O_L2;

		//81U
		P81U_L1.Parameter.Under		:= TRUE;
		P81U_L1.Parameter.Level		:= ProtPar.P81U_L1 * meter.Base.Fm;
		P81U_L1.Parameter.Time		:= ProtPar.T81U_L1;

		P81U_L2.Parameter.Under		:= TRUE;
		P81U_L2.Parameter.Level		:= ProtPar.P81U_L2 * meter.Base.Fm;
		P81U_L2.Parameter.Time		:= ProtPar.T81U_L2;

		//32OP
		P32OP_L1.Parameter.Under	:= FALSE;
		P32OP_L1.Parameter.Level	:= ProtPar.P32OP_L1 * meter.Base.Sm;
		P32OP_L1.Parameter.Time		:= ProtPar.T32OP_L1;

		//32UP
		P32UP_L1.Parameter.Under	:= TRUE;
		P32UP_L1.Parameter.Level	:= ProtPar.P32UP_L1 * meter.Base.Sm;
		P32UP_L1.Parameter.Time		:= ProtPar.T32UP_L1;

		//32OQ
		P32OQ_L1.Parameter.Under	:= FALSE;
		P32OQ_L1.Parameter.Level	:= ProtPar.P32OQ_L1 * meter.Base.Sm;
		P32OQ_L1.Parameter.Time		:= ProtPar.T32OQ_L1;

		//32UQ
		P32UQ_L1.Parameter.Under	:= TRUE;
		P32UQ_L1.Parameter.Level	:= ProtPar.P32UQ_L1 * meter.Base.Sm;
		P32UQ_L1.Parameter.Time		:= ProtPar.T32UQ_L1;

		//50P
		P50PA_L1.Parameter.Under	:= FALSE;
		P50PA_L1.Parameter.Level	:= ProtPar.P50P_L1 * meter.Base.Im;
		P50PA_L1.Parameter.Time		:= ProtPar.T50P_L1;

		P50PB_L1.Parameter := P50PC_L1.Parameter := P50PA_L1.Parameter;

		P50PA_L2.Parameter.Under	:= FALSE;
		P50PA_L2.Parameter.Level	:= ProtPar.P50P_L2 * meter.Base.Im;
		P50PA_L2.Parameter.Time		:= ProtPar.T50P_L2;

		P50PB_L2.Parameter := P50PC_L2.Parameter := P50PA_L2.Parameter;

		//50Q
		P50Q_L1.Parameter.Under		:= FALSE;
		P50Q_L1.Parameter.Level		:= ProtPar.P50Q_L1 * meter.Base.Im;
		P50Q_L1.Parameter.Time		:= ProtPar.T50Q_L1;

		P50Q_L2.Parameter.Under		:= FALSE;
		P50Q_L2.Parameter.Level		:= ProtPar.P50Q_L2 * meter.Base.Im;
		P50Q_L2.Parameter.Time		:= ProtPar.T50Q_L2;

		//50G
		P50G_L1.Parameter.Under		:= FALSE;
		P50G_L1.Parameter.Level		:= ProtPar.P50G_L1 * meter.Base.Im;
		P50G_L1.Parameter.Time		:= ProtPar.T50G_L1;

		P50G_L2.Parameter.Under		:= FALSE;
		P50G_L2.Parameter.Level		:= ProtPar.P50G_L2 * meter.Base.Im;
		P50G_L2.Parameter.Time		:= ProtPar.T50G_L2;

		//51V
		P51VA_L1.Parameter.Ipk		:= ProtPar.P51V_L1 * meter.Base.Im;
		P51VA_L1.Parameter.Td		:= ProtPar.T51V_L1;
		P51VA_L1.Parameter.Vnom		:= meter.Base.Um / SQRT(3.0);
		P51VA_L1.Parameter.Curve	:= REAL_TO_UINT(ProtPar.C51V_L1);

		P51VB_L1.Parameter := P51VC_L1.Parameter := P51VA_L1.Parameter;

		//51P
		P51PA_L1.Parameter.Ipk		:= ProtPar.P51P_L1 * meter.Base.Im;
		P51PA_L1.Parameter.Td		:= ProtPar.T51P_L1;
		P51PA_L1.Parameter.Vnom		:= 0.0;
		P51PA_L1.Parameter.Curve	:= REAL_TO_UINT(ProtPar.C51P_L1);

		P51PB_L1.Parameter := P51PC_L1.Parameter := P51PA_L1.Parameter;

		//51Q
		P51Q_L1.Parameter.Ipk		:= ProtPar.P51Q_L1 * meter.Base.Im;
		P51Q_L1.Parameter.Td		:= ProtPar.T51Q_L1;
		P51Q_L1.Parameter.Vnom		:= 0.0;
		P51Q_L1.Parameter.Curve		:= REAL_TO_UINT(ProtPar.C51Q_L1);

		//51G
		P51G_L1.Parameter.Ipk		:= ProtPar.P51G_L1 * meter.Base.Im;
		P51G_L1.Parameter.Td		:= ProtPar.T51G_L1;
		P51G_L1.Parameter.Vnom		:= 0.0;
		P51G_L1.Parameter.Curve		:= REAL_TO_UINT(ProtPar.C51G_L1);

		//24
		P24_L1.Parameter.HZnom		:= meter.Base.Fm;
		P24_L1.Parameter.Vnom		:= meter.Base.Um;
		P24_L1.Parameter.VHZ		:= ProtPar.P24_L1;
		P24_L1.Parameter.Time		:= ProtPar.T24_L1;

		//40
		P40_L1.Parameter.diameter	:= ProtPar.D40_L1;
		P40_L1.Parameter.Offset		:= ProtPar.O40_L1;
		P40_L1.Parameter.Time		:= ProtPar.T40_L1;

		P40_L2.Parameter.diameter	:= ProtPar.D40_L2;
		P40_L2.Parameter.Offset		:= ProtPar.O40_L2;
		P40_L2.Parameter.Time		:= ProtPar.T40_L2;
	END_IF;

END_PROGRAM
```

### Share.typ
```iecst
TYPE
	PgsCb52 : 	STRUCT
		di : PgsCb52DI;
		st : PgsCb52ST;
	END_STRUCT;
	PgsCb52DI : 	STRUCT
		opened : BOOL;
		closed : BOOL;
	END_STRUCT;
	PgsCb52ST : 	STRUCT
		status_fail : BOOL;
		opened : BOOL;
		closed : BOOL;
	END_STRUCT;
END_TYPE
```

### Program Logical/Kontrol/CB52/cb52 (IEC)

#### Variables.var
```iecst
VAR
	timer : TON;
END_VAR
```

#### Cyclic.st
```iecst
PROGRAM _CYCLIC

    CB52.st.closed  := CB52.di.closed;
    CB52.st.opened  := NOT CB52.di.closed;
    //Status Fail
    timer( IN := NOT(CB52.di.closed XOR CB52.di.opened), PT := T#3s );
	CB52.st.status_fail := timer.Q;

END_PROGRAM
```

### Program Logical/Kontrol/File/File (IEC)

#### Cyclic.st - Cyclic code
```iecst
PROGRAM _CYCLIC

    TagUpdate();

END_PROGRAM
```

#### Init.st - Init code
```iecst
PROGRAM _INIT
    TagManager(enable:=TRUE);

    TagUpdate.enable    := TRUE;
    TagUpdate.ident     := TagManager.ident;
    TagUpdate.FileName  := ADR('tags.xml');
END_PROGRAM
```

### Share.var
```iecst
VAR
	Event : UDINT;
END_VAR
```

### Program Logical/Kontrol/Event/Event

#### Variables.var
```iecst
VAR
	EventCreate : PgsEvtCreate;
	EventDelete : PgsEvtDelete;
	EventUpdate : PgsEvtUpdate;
END_VAR
(*Test*)
VAR
	test : REAL;
END_VAR
```

#### Main.st
```iecst
PROGRAM _INIT
    EventCreate.enable  := TRUE;        // Habilita o bloco que cria os eventos
    EventUpdate.enable  := TRUE;        // Habilita o bloco que gerencia a gravação dos eventos
    EventUpdate.file_sz := 1000000;     // Tamanho máximo de cada arquivo em bytes
    EventUpdate.max_sz  := 1000000000;  // Tamanho máximo que será utilizado no disco em bytes
    EventUpdate.time    := 86400;       // Tempo que o Bloco verifica o tamanho ocupado em disco e apaga arquivos antigos se necessário.
    TagManager(enable:=TRUE);

    //Register Parameters
    PgsTagStartNode     (TagManager.ident, ADR('evt'));
    PgsTagRegisterBOOL  (TagManager.ident, FALSE, ADR('read_config'),   EventUpdate.read_config);
    PgsTagRegisterBOOL  (TagManager.ident, FALSE, ADR('clear_history'), EventUpdate.clear_history);
    PgsTagRegisterUDINT (TagManager.ident, TRUE,  ADR('file_sz'),       EventUpdate.file_sz);
    PgsTagRegisterUDINT (TagManager.ident, TRUE,  ADR('max_sz'),        EventUpdate.max_sz);
    PgsTagRegisterREAL  (TagManager.ident, TRUE,  ADR('time'),          EventUpdate.time);
    //Test
    PgsTagRegisterREAL  (TagManager.ident, FALSE,  ADR('test'),         test);
    PgsTagEndNode       (TagManager.ident);//evt
    test := 1;
END_PROGRAM

PROGRAM _CYCLIC
        EventCreate( tagIdent := TagManager.ident );
        EventCreate.enable := FALSE;
        EventUpdate( ident := EventCreate.ident );
        Event := EventCreate.ident;
END_PROGRAM

PROGRAM _EXIT
    Event := 0;
    REPEAT
        EventDelete(
            enable  := TRUE,
            ident   := EventCreate.ident
        );
    UNTIL EventDelete.status <> PGS_EVT_ST_RUNNING
    END_REPEAT;
END_PROGRAM
```

Listed in the project but not available here: Logical/Global.typ, Logical/Global.var, Logical/MemTables.var, Logical/Libraries/Kontrol/PgsAuto/Constants.var, Logical/Libraries/Kontrol/PgsAuto/PGS_MDB_TO_REAL.st, Logical/Libraries/Kontrol/PgsAuto/PGS_REAL_TO_MDB.st, Logical/Libraries/Kontrol/PgsAuto/PGS_MDB_TO_DINT.st, Logical/Libraries/Kontrol/PgsAuto/PgsAlarme.st, Logical/Libraries/Kontrol/PgsAuto/PgsFiltro.st, Logical/Libraries/Kontrol/PgsAuto/PgsSobre.st, Logical/Libraries/Kontrol/PgsAuto/PgsEnergia.st, Logical/Comm/Share.typ, Logical/Comm/Share.var, Logical/Auto/Modbus/MDB_Types.typ, Logical/Auto/Modbus/MDB_Variables.var, Logical/Auto/Modbus/MDB_Status, Logical/Auto/Modbus/MDB_Alarme/Cyclic.st, Logical/Auto/Modbus/MDB_Medida, Logical/Auto/Modbus/MDB_Parametro, Logical/Auto/Modbus/MDB_CMD/LocalFunctions.fun, Logical/Kontrol/Protection/Share.typ, Logical/Kontrol/Protection/Local.var, Logical/Kontrol/CB52/Share.var, Logical/Kontrol/File/Share.var, Logical/Kontrol/File/File/Exit.st, Logical/Kontrol/File/File/Variables.var, Logical/Kontrol/File/File/Types.typ, Logical/Kontrol/Command
